// TIA Portal V19 export
DATA_BLOCK "Control_DB"   // DB2
{ S7_Optimized_Access := 'TRUE' }
// stored: MemoryReserve 100
   VAR
      Enable_Sequence : Bool;
      LightBarier_1 : Bool;
      LightBarier_2 : Bool;
      Enable_Drives : Bool;
      Conveyor_Speed : Real;
      "Step" : Int;
   END_VAR
BEGIN
END_DATA_BLOCK
